FUNCTION_BLOCK sequence_E_04_AX_SR (* Sequence with 4 Outputs, Transition by EVENT, with AX Adapter, STOP (safety off) and RESUME Events *)
  (* Standard: 61499-2; Description: Copyright (c) 2024 HR Agrartechnik GmbH This program and the accompanying materials are made available under the terms of the Eclipse Public License 2.0 which is available at https://www.eclipse.org/legal/epl-2.0/ SPDX-License-Identifier: EPL-2.0 *)
  (* Version 1.1, 2026-02-23, Franz Höpfinger, HR Agrartechnik GmbH *)
  PACKAGE logiBUS::utils::sequence::event;
  IMPORT logiBUS::utils::sequence::const::sequence;
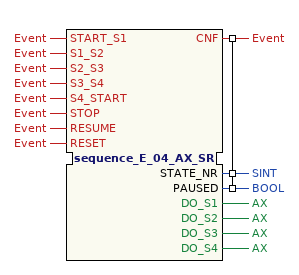
  EVENT_INPUT
    START_S1; (* jump from START to State_01 *)
    S1_S2; (* jump from State_01 to State_02 *)
    S2_S3; (* jump from State_02 to State_03 *)
    S3_S4; (* jump from State_03 to State_04 *)
    S4_START; (* jump from State_04 to START *)
    STOP; (* Stop current state immediately - ALL outputs go OFF (dead-man stop) *)
    RESUME; (* Resume from pause - continue with current state *)
    RESET; (* Reset from any State to START *)
  END_EVENT
  EVENT_OUTPUT
    CNF WITH STATE_NR, PAUSED; (* Execution Confirmation *)
  END_EVENT
  VAR_OUTPUT
    STATE_NR : SINT; (* State Number, START = 0, State_01 = 1 and so on. *)
    PAUSED : BOOL; (* TRUE if sequencer is paused (STOP active) *)
  END_VAR
  PLUGS
    DO_S1 : adapter::types::unidirectional::AX; (* Output if State_01 is active *)
    DO_S2 : adapter::types::unidirectional::AX; (* Output if State_02 is active *)
    DO_S3 : adapter::types::unidirectional::AX; (* Output if State_03 is active *)
    DO_S4 : adapter::types::unidirectional::AX; (* Output if State_04 is active *)
  END_PLUGS
  VAR
    savedState : SINT; (* Store current state when paused *)
  END_VAR
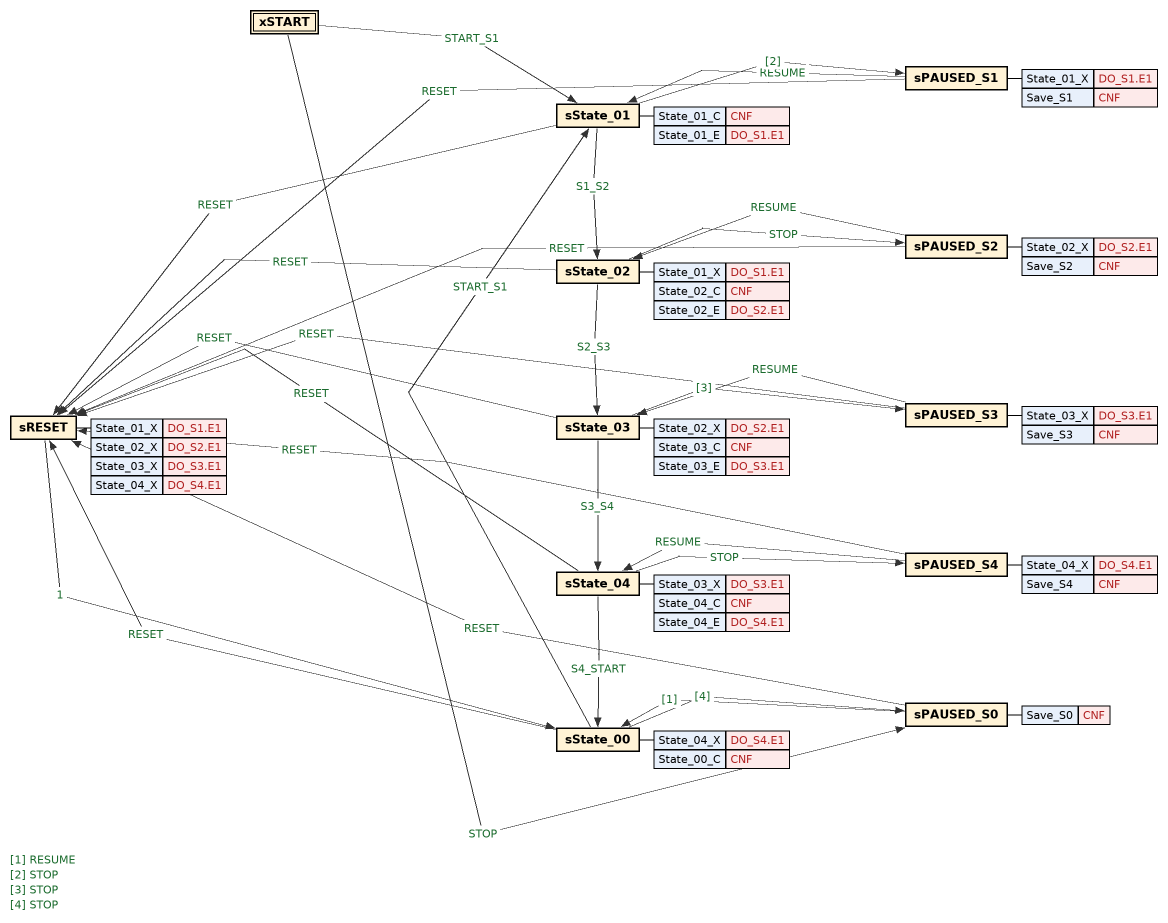
  EC_STATES
    xSTART; (* Initial State *)
    sState_01 : State_01_C -> CNF, State_01_E -> DO_S1.E1;
    sState_02 : State_01_X -> DO_S1.E1, State_02_C -> CNF, State_02_E -> DO_S2.E1;
    sState_03 : State_02_X -> DO_S2.E1, State_03_C -> CNF, State_03_E -> DO_S3.E1;
    sState_04 : State_03_X -> DO_S3.E1, State_04_C -> CNF, State_04_E -> DO_S4.E1;
    sState_00 : State_04_X -> DO_S4.E1, State_00_C -> CNF;
    sPAUSED_S1 : State_01_X -> DO_S1.E1, Save_S1 -> CNF; (* Paused while in State_01 - Output OFF *)
    sPAUSED_S2 : State_02_X -> DO_S2.E1, Save_S2 -> CNF; (* Paused while in State_02 - Output OFF *)
    sPAUSED_S3 : State_03_X -> DO_S3.E1, Save_S3 -> CNF; (* Paused while in State_03 - Output OFF *)
    sPAUSED_S4 : State_04_X -> DO_S4.E1, Save_S4 -> CNF; (* Paused while in State_04 - Output OFF *)
    sPAUSED_S0 : Save_S0 -> CNF; (* Paused while in START/State_00 - Output OFF *)
    sRESET : State_01_X -> DO_S1.E1, State_02_X -> DO_S2.E1, State_03_X -> DO_S3.E1, State_04_X -> DO_S4.E1;
  END_STATES
  EC_TRANSITIONS
    sState_01 TO sState_02 := S1_S2;
    sState_02 TO sState_03 := S2_S3;
    sState_03 TO sState_04 := S3_S4;
    sState_00 TO sState_01 := START_S1;
    sState_04 TO sState_00 := S4_START;
    xSTART TO sState_01 := START_S1;
    sState_01 TO sPAUSED_S1 := STOP;
    sState_02 TO sPAUSED_S2 := STOP;
    sState_03 TO sPAUSED_S3 := STOP;
    sState_04 TO sPAUSED_S4 := STOP;
    sState_00 TO sPAUSED_S0 := STOP;
    xSTART TO sPAUSED_S0 := STOP;
    sPAUSED_S1 TO sState_01 := RESUME;
    sPAUSED_S2 TO sState_02 := RESUME;
    sPAUSED_S3 TO sState_03 := RESUME;
    sPAUSED_S4 TO sState_04 := RESUME;
    sPAUSED_S0 TO sState_00 := RESUME;
    sState_01 TO sRESET := RESET;
    sState_02 TO sRESET := RESET;
    sState_03 TO sRESET := RESET;
    sState_04 TO sRESET := RESET;
    sState_00 TO sRESET := RESET;
    sPAUSED_S1 TO sRESET := RESET;
    sPAUSED_S2 TO sRESET := RESET;
    sPAUSED_S3 TO sRESET := RESET;
    sPAUSED_S4 TO sRESET := RESET;
    sPAUSED_S0 TO sRESET := RESET;
    sRESET TO sState_00 := 1;
  END_TRANSITIONS
  ALGORITHM State_00_C IN ST:
 // State_00 Confirmation Step
STATE_NR := sequence::State_00;
PAUSED := BOOL#FALSE;
savedState := sequence::State_00;
  END_ALGORITHM
  ALGORITHM State_01_C IN ST:
 // State_01 Confirmation Step
STATE_NR := sequence::State_01;
PAUSED := BOOL#FALSE;
savedState := sequence::State_01;
  END_ALGORITHM
  ALGORITHM State_02_C IN ST:
 // State_02 Confirmation Step
STATE_NR := sequence::State_02;
PAUSED := BOOL#FALSE;
savedState := sequence::State_02;
  END_ALGORITHM
  ALGORITHM State_03_C IN ST:
 // State_03 Confirmation Step
STATE_NR := sequence::State_03;
PAUSED := BOOL#FALSE;
savedState := sequence::State_03;
  END_ALGORITHM
  ALGORITHM State_04_C IN ST:
 // State_04 Confirmation Step
STATE_NR := sequence::State_04;
PAUSED := BOOL#FALSE;
savedState := sequence::State_04;
  END_ALGORITHM
  ALGORITHM Save_S0 IN ST:
 // Pause in State_00
STATE_NR := savedState;
PAUSED := BOOL#TRUE;
  END_ALGORITHM
  ALGORITHM Save_S1 IN ST:
 // Pause in State_01
STATE_NR := savedState;
PAUSED := BOOL#TRUE;
  END_ALGORITHM
  ALGORITHM Save_S2 IN ST:
 // Pause in State_02
STATE_NR := savedState;
PAUSED := BOOL#TRUE;
  END_ALGORITHM
  ALGORITHM Save_S3 IN ST:
 // Pause in State_03
STATE_NR := savedState;
PAUSED := BOOL#TRUE;
  END_ALGORITHM
  ALGORITHM Save_S4 IN ST:
 // Pause in State_04
STATE_NR := savedState;
PAUSED := BOOL#TRUE;
  END_ALGORITHM
  ALGORITHM State_01_E IN ST:
 // State_01 Entry Step
DO_S1.D1 := BOOL#TRUE; // ON
  END_ALGORITHM
  ALGORITHM State_01_X IN ST:
 // State_01 Exit Step
DO_S1.D1 := BOOL#FALSE;
  END_ALGORITHM
  ALGORITHM State_02_E IN ST:
 // State_02 Entry Step
DO_S2.D1 := BOOL#TRUE; // ON
  END_ALGORITHM
  ALGORITHM State_02_X IN ST:
 // State_02 Exit Step
DO_S2.D1 := BOOL#FALSE;
  END_ALGORITHM
  ALGORITHM State_03_E IN ST:
 // State_03 Entry Step
DO_S3.D1 := BOOL#TRUE; // ON
  END_ALGORITHM
  ALGORITHM State_03_X IN ST:
 // State_03 Exit Step
DO_S3.D1 := BOOL#FALSE;
  END_ALGORITHM
  ALGORITHM State_04_E IN ST:
 // State_04 Entry Step
DO_S4.D1 := BOOL#TRUE; // ON
  END_ALGORITHM
  ALGORITHM State_04_X IN ST:
 // State_04 Exit Step
DO_S4.D1 := BOOL#FALSE;
  END_ALGORITHM
END_FUNCTION_BLOCK
